Fanuc KAREL source: MSG_CONNECT.kl

PROGRAM T
%NOLOCKGROUP
VAR
 v0 : STRING[40]
 v1 : INTEGER
BEGIN
 MSG_CONNECT(v0, v1)
END T
